// Mitsubishi GX Works2 project: 240409_지연동작_한시복귀회로   PLC: Q03UDV

PROGRAM MAIN
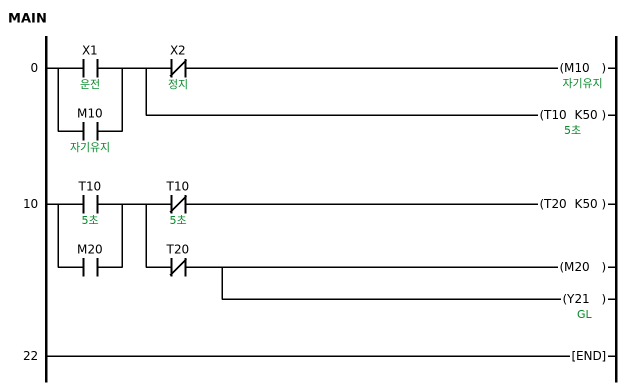
0     LD      X1  ; 운전
      OR      M10  ; 자기유지
      MPS
      ANI     X2  ; 정지
      OUT     M10  ; 자기유지
      MPP
      OUT     T10 K50  ; 5초
10    LD      T10  ; 5초
      OR      M20
      MPS
      ANI     T10  ; 5초
      OUT     T20 K50
      MPP
      ANI     T20
      OUT     M20
      OUT     Y21  ; GL
22    END
END_PROGRAM

// device comments not shown above
X0  ; 정지
Y22  ; 정지
